{attribute addProperty BoxType "CU1128-0000-0001"}
{attribute addProperty Id "A_0006_CU1128_0000_0002A_0006_CU1128_0000_0002_C9ADC9BE928116A_0005_CU1128_0000_0001_2_CU1128_BCU1128_179A0949162A_0005_CU1128_0000_0001_3_CU1128_CCU1128_179A0949162"}
{attribute addProperty CRC "3504570307"}
{attribute addProperty SizeInBites "960"}
{attribute addProperty SizeInBytes "120"}
TYPE A_0005_CU1128_0000_0001_D0E37FC3 EXTENDS CU1128_179A0949 :
STRUCT
	{attribute addProperty Name "A_0006_CU1128_0000_0002"}
	A_0006_CU1128_0000_0002 : A_0006_CU1128_0000_0002_C9ADC9BE;
	{attribute addProperty Name "A_0005_CU1128_0000_0001_2_CU1128_B"}
	A_0005_CU1128_0000_0001_2_CU1128_B : CU1128_179A0949;
	{attribute addProperty Name "A_0005_CU1128_0000_0001_3_CU1128_C"}
	A_0005_CU1128_0000_0001_3_CU1128_C : CU1128_179A0949;
END_STRUCT
END_TYPE

(* stored: Version 1.2.0.0, ProductVersion 3.1.4024.9
   DUT A_0005_CU1128_0000_0001_D0E37FC3: Id {fddfe367-c7b2-4935-a308-35b33c182e8a} *)
